// TwinCAT 3 PLC project SPS1
// ProgramVersion: 3.1.4023.0
// libraries:
//   Tc2_MC2, * (Beckhoff Automation GmbH)
//   Tc2_Standard, * (Beckhoff Automation GmbH)
//   Tc2_System, * (Beckhoff Automation GmbH)
//   Tc3_Module, * (Beckhoff Automation GmbH)
//   VisuSymbols,3.5.10.0,System
// project tree:
//   / GlobalTextList.TcGTLO, PlcTask.TcTTO, Visualisierungsmanager.TcVMO (not stored)
//   GVLs/ GVL.TcGVL
//   POUs/ Achse1.TcPOU, MAIN.TcPOU
//   VISUs/ Visualization.TcVIS
// real-time tasks:
//   TASK PlcTask: cycle T#10ms, priority 20, ADS port 350
// motion (NC):
//   TASK NC-Task 1 SAF: cycle T#2ms, priority 4, ADS port 501
//   TASK NC-Task 1 SVB: cycle T#10ms, priority 8, ADS port 511
//   AXIS Achse 1 Blau (id 1)
//     OtherSettings: AllowMotionCmdToSlave=true
//     encoder EncType=1
//     drive DrvType=5
//       Analog: TorqueSetpointScale=10, ScaleFactorActTorque=0.1
//       TimeComp: TaskDelayCycles=1
//     controller CtrType=1
//       CtrPara: PriorControlFactor=1
//         Observer: BandWidth=20
//   AXIS Achse 2 Rot (id 2)
//     OtherSettings: AllowMotionCmdToSlave=true
//     encoder EncType=1
//     drive DrvType=5
//       Analog: TorqueSetpointScale=10, ScaleFactorActTorque=0.1
//     controller CtrType=1
//       CtrPara: PriorControlFactor=1
//         Observer: BandWidth=20
// variable links:
//   SPS1/SPS1 Instance <-> NC-Task 1 SAF/Axes/Achse 1 Blau
//     PlcTask Inputs/GVL.Achse1_Ref.NcToPlc <-> Outputs/ToPlc
//     PlcTask Outputs/GVL.Achse1_Ref.PlcToNc <-> Inputs/FromPlc
//   SPS1/SPS1 Instance <-> NC-Task 1 SAF/Axes/Achse 2 Rot
//     PlcTask Inputs/GVL.Achse2_Ref.NcToPlc <-> Outputs/ToPlc
//     PlcTask Outputs/GVL.Achse2_Ref.PlcToNc <-> Inputs/FromPlc

CONFIGURATION SPS1
    RESOURCE PLC ON TwinCAT3
        TASK PlcTask(INTERVAL := T#10ms, PRIORITY := 20);
        PROGRAM MAIN WITH PlcTask : MAIN;
    END_RESOURCE
END_CONFIGURATION

// ---- GVLs/GVL.TcGVL
{attribute 'qualified_only'}
VAR_GLOBAL
	Achse2_Ref: AXIS_REF;
	Achse1_Ref: AXIS_REF;
END_VAR

// ---- POUs/MAIN.TcPOU
PROGRAM MAIN
VAR
	A1: Achse1;
END_VAR

A1();

END_PROGRAM

// ---- POUs/Achse1.TcPOU
FUNCTION_BLOCK Achse1
VAR
	MC_Power_1: MC_POWER;
	MC_Move1: MC_MoveRelative;
END_VAR

MC_Move1(Axis := GVL.Achse1_Ref, Distance := 250, Velocity := 200, Acceleration := 50, Deceleration := 50); // MC_MoveRelative
MC_Power_1(Axis := GVL.Achse1_Ref, Enable := 1, Enable_Positive := 1, Enable_Negative := 1, Override := 50); // MC_POWER

END_FUNCTION_BLOCK

// ---- VISUs/Visualization.TcVIS
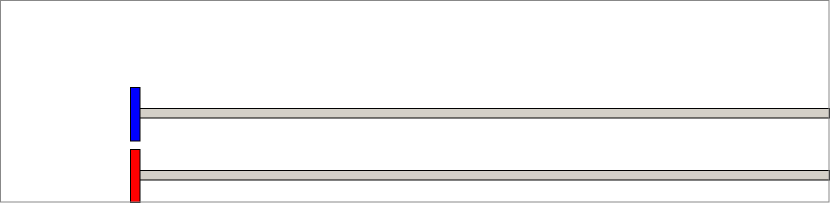
VISUALIZATION Visualization  // 830x203
    Rectangle (130,108 700x10)
    Rectangle (130,87 10x54)
        p3560616238: GVL.Achse1_Ref.NcToPlc.ActPos
    Rectangle (130,170 700x10)
    Rectangle (130,149 10x54)
        p3560616238: GVL.Achse2_Ref.NcToPlc.ActPos
END_VISUALIZATION
